FUNCTION alg_a_transfer2droppos : BOOL
VAR_INPUT
	state: STATE;
END_VAR

alg_a_transfer2droppos := FALSE;

END_FUNCTION

(* stored: Version 1.1.0.1, ProductVersion 3.1.4022.18
   POU alg_a_transfer2droppos: Id {d112ac19-ab66-4cb5-ad4c-3e0871fec062}, SpecialFunc None *)
